(* PLC project Sin nombre, Desconocido Sin nombre 1 *)
(* stored: creationDateTime 2024-03-26T11:05:44, modificationDateTime 2024-03-30T18:16:12 *)

(* B *)
PROGRAM program0
  VAR
    A AT %IX0.0 : BOOL;
    B AT %IX0.1 : BOOL;
    C AT %IX0.2 : BOOL;
    H1 AT %QX0.0 : BOOL;
    H2 AT %QX0.1 : BOOL;
    H3 AT %QX0.2 : BOOL;
    H4 AT %QX0.3 : BOOL;
    H5 AT %QX0.4 : BOOL;
  END_VAR

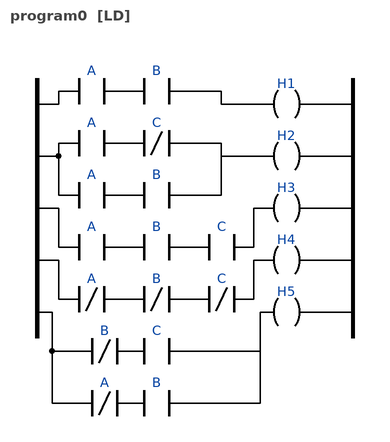
(* LD diagram, written out as Structured Text *)
H1 := A AND B;
H2 := A AND (NOT C OR B);
H3 := A AND B AND C;
H4 := NOT A AND NOT B AND NOT C;
H5 := NOT B AND C OR NOT A AND B;
END_PROGRAM

CONFIGURATION Config0
  RESOURCE Res0 ON PLC
    TASK task0(INTERVAL := T#20ms, PRIORITY := 0);
    PROGRAM instance0 WITH task0 : program0;
  END_RESOURCE
END_CONFIGURATION
